{attribute 'qualified_only'}
{attribute 'strict'}
{attribute 'to_string'}
TYPE E_State_RobotGeneral :
(
	Init := 0,
	AutoEnable,
	OperationEnable,
	Error,
	ErrorReset,
	ServoOn,
	Start,
	Started,
	ProgramStop,
	ProgramReset
	
);
END_TYPE

(* stored: Version 1.1.0.1, ProductVersion 3.1.4024.11
   DUT E_State_RobotGeneral: Id {ebfe3363-1056-42c1-aa6f-6522c1238922} *)
